(* IEC 61131-3 sources: MyTestRepos/BATTERY/PRG (part 2) *)

(* ---- PRG_DO.st ---- *)
PROGRAM PRG_DO
VAR
	F_Trig : ARRAY[1..cnst_num_do] OF F_TRIG;
	i: INT;
	ManualFixChannels : BOOL; (*Will reset channels if faulty, i.e. card number is zero*)
	Reset: BOOL;
	Firstrun: BOOL;
	(*Interal variables*)
	Fan_SR : 				SR;

	(* Digital Outputs*)
	do_RunningLamp: str_DoProcess;
	do_Running: str_DoProcess;
	do_StoppedLamp: str_DoProcess;
	do_Stopped: str_DoProcess;
	do_FaultLamp: str_DoProcess;
	do_WarningLamp: str_DoProcess;
	do_StartFan: str_DoProcess;
	do_EnergizedLamp: str_DoProcess;
	do_LampTest: str_DoProcess;
	do_ReadyLamp: str_DoProcess;
	do_ChargingLamp: str_DoProcess;
	do_ShutdownPlcFailure: str_DoProcess;
	do_LocalLamp: str_DoProcess;

	do_RunningLamp_daemon: fb_DoProcess;
	do_Running_daemon: fb_DoProcess;
	do_StoppedLamp_daemon: fb_DoProcess;
	do_Stopped_daemon: fb_DoProcess;
	do_FaultLamp_daemon: fb_DoProcess;
	do_WarningLamp_daemon: fb_DoProcess;
	do_StartFan_daemon: fb_DoProcess;
	do_EnergizedLamp_daemon: fb_DoProcess;
	do_LampTest_daemon: fb_DoProcess;
	do_ReadyLamp_daemon: fb_DoProcess;
	do_ChargingLamp_daemon: fb_DoProcess;
	do_ShutdownPlcFailure_daemon: fb_DoProcess;
	do_LocalLamp_daemon: fb_DoProcess;
END_VAR

VAR RETAIN
	do_RunningLamp_setup: str_DoSetup;
	do_Running_setup: str_DoSetup;
	do_StoppedLamp_setup: str_DoSetup;
	do_Stopped_setup: str_DoSetup;
	do_FaultLamp_setup: str_DoSetup;
	do_WarningLamp_setup: str_DoSetup;
	do_StartFan_setup: str_DoSetup;
	do_EnergizedLamp_setup: str_DoSetup;
	do_LampTest_setup: str_DoSetup;
	do_ReadyLamp_setup: str_DoSetup;
	do_ChargingLamp_setup: str_DoSetup;
	do_ShutdownPlcFailure_setup: str_DoSetup;
	do_LocalLamp_setup: str_DoSetup;
END_VAR

Reset := PRG_Functions.Reset;

(*Setup the HMI variables so that they are equal to actual used variables*)
IF (NOT Firstrun) THEN
	hmi_DoSetup[1]:=do_RunningLamp_setup;
	hmi_DoSetup[2]:=do_Running_setup;
	hmi_DoSetup[3]:=do_StoppedLamp_setup;
	hmi_DoSetup[4]:=do_Stopped_setup;
	hmi_DoSetup[5]:=do_FaultLamp_setup;
	hmi_DoSetup[6]:=do_WarningLamp_setup;
	hmi_DoSetup[7]:=do_StartFan_setup;
	hmi_DoSetup[8]:=do_EnergizedLamp_setup;
	hmi_DoSetup[9]:=do_LampTest_setup;
	hmi_DoSetup[10]:=do_ReadyLamp_setup;
	hmi_DoSetup[11]:=do_ChargingLamp_setup;
	hmi_DoSetup[12]:=do_ShutdownPlcFailure_setup;
	hmi_DoSetup[13]:=do_LocalLamp_setup;
	Firstrun := TRUE;
END_IF

do_StartFan_daemon (setup:=do_StartFan_setup,inPV:=do_StartFan);
do_LampTest_daemon (setup:=do_LampTest_setup,inPV:=do_LampTest);
do_Running_daemon (setup:=do_Running_setup,inPV:=do_Running);
do_Stopped_daemon (setup:=do_Stopped_setup,inPV:=do_Stopped);
do_ShutdownPlcFailure_daemon (setup:=do_ShutdownPlcFailure_setup,inPV:=do_ShutdownPlcFailure);

IF PRG_HMI.DoorSettings.enRunningLamp THEN
	do_RunningLamp_daemon (setup:=do_RunningLamp_setup,inPV:=do_RunningLamp);
END_IF

IF PRG_HMI.DoorSettings.enStoppedLamp THEN
	do_StoppedLamp_daemon (setup:=do_StoppedLamp_setup,inPV:=do_StoppedLamp);
END_IF

IF PRG_HMI.DoorSettings.enFaultLamp THEN
	do_FaultLamp_daemon (setup:=do_FaultLamp_setup,inPV:=do_FaultLamp);
END_IF

IF PRG_HMI.DoorSettings.enWarningLamp THEN
	do_WarningLamp_daemon (setup:=do_WarningLamp_setup,inPV:=do_WarningLamp);
END_IF

IF PRG_HMI.DoorSettings.enChargingLamp THEN
	do_ChargingLamp_daemon (setup:=do_ChargingLamp_setup,inPV:=do_ChargingLamp);
END_IF

IF PRG_HMI.DoorSettings.enLocalLamp THEN
	do_LocalLamp_daemon (setup:=do_LocalLamp_setup,inPV:=do_LocalLamp);
END_IF

IF PRG_HMI.DoorSettings.enReadyLamp THEN
	do_ReadyLamp_daemon (setup:=do_ReadyLamp_setup,inPV:=do_ReadyLamp);
END_IF

IF PRG_HMI.DoorSettings.enEnergizedLamp THEN
	do_EnergizedLamp_daemon (setup:=do_EnergizedLamp_setup,inPV:=do_EnergizedLamp);
END_IF

hmi_DoPV[1]:=do_RunningLamp_daemon.inPV;
hmi_DoPV[2]:=do_Running_daemon.inPV;
hmi_DoPV[3]:=do_StoppedLamp_daemon.inPV;
hmi_DoPV[4]:=do_Stopped_daemon.inPV;
hmi_DoPV[5]:=do_FaultLamp_daemon.inPV;
hmi_DoPV[6]:=do_WarningLamp_daemon.inPV;
hmi_DoPV[7]:=do_StartFan_daemon.inPV;
hmi_DoPV[8]:=do_EnergizedLamp_daemon.inPV;
hmi_DoPV[9]:=do_LampTest_daemon.inPV;
hmi_DoPV[10]:=do_ReadyLamp_daemon.inPV;
hmi_DoPV[11]:=do_ChargingLamp_daemon.inPV;
hmi_DoPV[12]:=do_ShutdownPlcFailure_daemon.inPV;
hmi_DoPV[13]:=do_LocalLamp_daemon.inPV;

IF (ManualFixChannels) THEN  (*If manually forced: re-configure the channels*)
	FOR i:=0 TO cnst_num_do BY 1 DO				(*Check if channel info is empty and restore if so.*)
		IF (hmi_DoSetup[i].CardNb = 0 AND PRG_HMI.setup_DioCard1_Number <> 0) THEN
			hmi_RestoreDefault_do[i] := TRUE;
		END_IF
	END_FOR;
	ManualFixChannels := FALSE;
END_IF

(*------------------------------------Control of cabinet lamps -------------------------------------*)

(*In Local Lamp*)
IF PRG_HMI.DoorSettings.enLocalLamp THEN
	IF(PRG_IAS.IasCommunication.Alarm AND (PRG_Operation.ControlPlace.ctrlLocation = e_Remote)) THEN
		do_LocalLamp.PV := PRG_StateMain.LedBlinker.CLK_Pulse;
	ELSE
		do_LocalLamp.PV	:= PRG_Operation.ControlPlace.ctrlLocation = e_Local XOR PRG_HMI.LamptestPulsetrain.CLK_Pulse;
	END_IF
END_IF

(*Running Lamp*)
IF PRG_HMI.DoorSettings.enRunningLamp THEN
	do_RunningLamp.PV := (PRG_StateMain.RunningLamp XOR PRG_HMI.LamptestPulsetrain.CLK_Pulse);
END_IF

(*Stopped Lamp*)
IF PRG_HMI.DoorSettings.enStoppedLamp THEN
	do_StoppedLamp.PV := (PRG_StateMain.StoppedLamp XOR PRG_HMI.LamptestPulsetrain.CLK_Pulse );
END_IF

(*Warning Lamp*)
IF PRG_HMI.DoorSettings.enWarningLamp THEN
	do_WarningLamp.PV := (PRG_Alarms.Repeat_Alarm.Alarm_common XOR PRG_HMI.LamptestPulsetrain.CLK_Pulse);
END_IF

(*Fault Lamp*)
IF PRG_HMI.DoorSettings.enFaultLamp THEN
	do_FaultLamp.PV := (PRG_Faults.Repeat_Fault.Alarm_common XOR PRG_HMI.LamptestPulsetrain.CLK_Pulse);
END_IF

(*Charging Lamp*)
IF PRG_HMI.DoorSettings.enChargingLamp THEN
	do_ChargingLamp.PV := (PRG_Battery.batteryCharging XOR PRG_HMI.LamptestPulsetrain.CLK_Pulse);
END_IF

(*Ready to Start Lamp*)
IF PRG_HMI.DoorSettings.enReadyLamp THEN
	do_ReadyLamp.PV := (PRG_HMI.ReadyToStart XOR PRG_HMI.LamptestPulsetrain.CLK_Pulse);
END_IF

(*Energized Lamp*)
IF PRG_HMI.DoorSettings.enEnergizedLamp THEN
	do_EnergizedLamp.PV := (PRG_Battery.BatteryMinOneConnected XOR PRG_HMI.LamptestPulsetrain.CLK_Pulse);
END_IF

(*Lamp test relay for lamps not connected to PLC*)
do_LampTest.PV := PRG_HMI.LamptestPulsetrain.CLK_Pulse;

(*------------------------------------Hardwire Status Outputs -------------------------------------*)

do_Stopped.PV := PRG_StateMain.StoppedOutput;
do_Running.PV := PRG_StateMain.RunningOutput;

(*------------------------------------Control of cabinet fan -------------------------------------*)
Fan_SR(
	SET1 := PRG_AI.ai_CabinetTemperature.Level.H,
	RESET := PRG_AI.ai_CabinetTemperature.Level.L,
	Q1 => do_StartFan.PV
);

(*------------------------------------ Hardwire Shutdown -------------------------------------*)
(*If modbus fault or no stopping - drop the white gloves.*)
IF 	(PRG_BatteryComm.CorvusBMS_Total_Comm_Fault OR PRG_StateMain.stoppingTON.Q OR PRG_Drive.CommFault[1]) THEN
	do_ShutdownPlcFailure.PV := FALSE;
ELSE
	do_ShutdownPlcFailure.PV := TRUE;
END_IF

END_PROGRAM

ACTIONS

ACTION Settings

(**************do_RunningLamp***********************)
IF (RestoreAllToDefault OR do_RunningLamp_setup.RestoreDefault  OR hmi_RestoreDefault_do[1]) THEN
	do_RunningLamp_setup.Name:='do_RunningLamp';
	do_RunningLamp_setup.CardNb:=PRG_HMI.setup_DioCard1_Number;
	do_RunningLamp_setup.ChannelMode:=2;
	do_RunningLamp_setup.ChannelNb:=1;
	do_RunningLamp_setup.Enable.Forcing:=0;
	do_RunningLamp_setup.Levels.ForceValue:=0;
END_IF
IF (hmi_RestoreDefault_do[1] OR RestoreAllToDefault OR do_RunningLamp_setup.RestoreDefault) THEN (*Copy values into HMI variable and reset*)
	hmi_DoSetup[1]:=do_RunningLamp_setup; (*Copy setup values from retain into hmi variable*)
	hmi_RestoreDefault_do[1]:=FALSE; (*Make sure that the restore variable is turned off after one restore command*)
	do_RunningLamp_setup.RestoreDefault:=FALSE; (*Make sure that the restore variable is turned off after one restore command*)
END_IF
IF (hmi_DoWriteSetup[1]) THEN
	do_RunningLamp_setup:=hmi_DoSetup[1]; (*Paste hmi changes back into setup variable*)
	hmi_DoWriteSetup[1]:=FALSE; (*Make sure that the write variable is turned off after one write command*)
END_IF
F_Trig[1](CLK:=hmi_DoPV[1].IsForced); (*Reset HMI forcing dialog when timer runs out*)
IF (F_Trig[1].Q) THEN hmi_DoSetup[1].Enable.Forcing:=FALSE;do_RunningLamp_setup.Enable.Forcing:=FALSE; END_IF
(**************************************************)

(**************do_Running***********************)
IF (RestoreAllToDefault OR do_Running_setup.RestoreDefault  OR hmi_RestoreDefault_do[2]) THEN
	do_Running_setup.Name:='do_Running';
	do_Running_setup.CardNb:=PRG_HMI.setup_DioCard1_Number;
	do_Running_setup.ChannelMode:=2;
	do_Running_setup.ChannelNb:=2;
	do_Running_setup.Enable.Forcing:=0;
	do_Running_setup.Levels.ForceValue:=0;
END_IF
IF (hmi_RestoreDefault_do[2] OR RestoreAllToDefault OR do_Running_setup.RestoreDefault) THEN (*Copy values into HMI variable and reset*)
	hmi_DoSetup[2]:=do_Running_setup; (*Copy setup values from retain into hmi variable*)
	hmi_RestoreDefault_do[2]:=FALSE; (*Make sure that the restore variable is turned off after one restore command*)
	do_Running_setup.RestoreDefault:=FALSE; (*Make sure that the restore variable is turned off after one restore command*)
END_IF
IF (hmi_DoWriteSetup[2]) THEN
	do_Running_setup:=hmi_DoSetup[2]; (*Paste hmi changes back into setup variable*)
	hmi_DoWriteSetup[2]:=FALSE; (*Make sure that the write variable is turned off after one write command*)
END_IF
F_Trig[2](CLK:=hmi_DoPV[2].IsForced); (*Reset HMI forcing dialog when timer runs out*)
IF (F_Trig[2].Q) THEN hmi_DoSetup[2].Enable.Forcing:=FALSE;do_Running_setup.Enable.Forcing:=FALSE; END_IF
(**************************************************)

(**************do_StoppedLamp***********************)
IF (RestoreAllToDefault OR do_StoppedLamp_setup.RestoreDefault  OR hmi_RestoreDefault_do[3]) THEN
	do_StoppedLamp_setup.Name:='do_StoppedLamp';
	do_StoppedLamp_setup.CardNb:=PRG_HMI.setup_DioCard1_Number;
	do_StoppedLamp_setup.ChannelMode:=2;
	do_StoppedLamp_setup.ChannelNb:=3;
	do_StoppedLamp_setup.Enable.Forcing:=0;
	do_StoppedLamp_setup.Levels.ForceValue:=0;
END_IF
IF (hmi_RestoreDefault_do[3] OR RestoreAllToDefault OR do_StoppedLamp_setup.RestoreDefault) THEN (*Copy values into HMI variable and reset*)
	hmi_DoSetup[3]:=do_StoppedLamp_setup; (*Copy setup values from retain into hmi variable*)
	hmi_RestoreDefault_do[3]:=FALSE; (*Make sure that the restore variable is turned off after one restore command*)
	do_StoppedLamp_setup.RestoreDefault:=FALSE; (*Make sure that the restore variable is turned off after one restore command*)
END_IF
IF (hmi_DoWriteSetup[3]) THEN
	do_StoppedLamp_setup:=hmi_DoSetup[3]; (*Paste hmi changes back into setup variable*)
	hmi_DoWriteSetup[3]:=FALSE; (*Make sure that the write variable is turned off after one write command*)
END_IF
F_Trig[3](CLK:=hmi_DoPV[3].IsForced); (*Reset HMI forcing dialog when timer runs out*)
IF (F_Trig[3].Q) THEN hmi_DoSetup[3].Enable.Forcing:=FALSE;do_StoppedLamp_setup.Enable.Forcing:=FALSE; END_IF
(**************************************************)

(**************do_Stopped***********************)
IF (RestoreAllToDefault OR do_Stopped_setup.RestoreDefault  OR hmi_RestoreDefault_do[4]) THEN
	do_Stopped_setup.Name:='do_Stopped';
	do_Stopped_setup.CardNb:=PRG_HMI.setup_DioCard1_Number;
	do_Stopped_setup.ChannelMode:=2;
	do_Stopped_setup.ChannelNb:=4;
	do_Stopped_setup.Enable.Forcing:=0;
	do_Stopped_setup.Levels.ForceValue:=0;
END_IF
IF (hmi_RestoreDefault_do[4] OR RestoreAllToDefault OR do_Stopped_setup.RestoreDefault) THEN (*Copy values into HMI variable and reset*)
	hmi_DoSetup[4]:=do_Stopped_setup; (*Copy setup values from retain into hmi variable*)
	hmi_RestoreDefault_do[4]:=FALSE; (*Make sure that the restore variable is turned off after one restore command*)
	do_Stopped_setup.RestoreDefault:=FALSE; (*Make sure that the restore variable is turned off after one restore command*)
END_IF
IF (hmi_DoWriteSetup[4]) THEN
	do_Stopped_setup:=hmi_DoSetup[4]; (*Paste hmi changes back into setup variable*)
	hmi_DoWriteSetup[4]:=FALSE; (*Make sure that the write variable is turned off after one write command*)
END_IF
F_Trig[4](CLK:=hmi_DoPV[4].IsForced); (*Reset HMI forcing dialog when timer runs out*)
IF (F_Trig[4].Q) THEN hmi_DoSetup[4].Enable.Forcing:=FALSE;do_Stopped_setup.Enable.Forcing:=FALSE; END_IF
(**************************************************)

(**************do_FaultLamp***********************)
IF (RestoreAllToDefault OR do_FaultLamp_setup.RestoreDefault  OR hmi_RestoreDefault_do[5]) THEN
	do_FaultLamp_setup.Name:='do_FaultLamp';
	do_FaultLamp_setup.CardNb:=PRG_HMI.setup_DioCard1_Number;
	do_FaultLamp_setup.ChannelMode:=2;
	do_FaultLamp_setup.ChannelNb:=5;
	do_FaultLamp_setup.Enable.Forcing:=0;
	do_FaultLamp_setup.Levels.ForceValue:=0;
END_IF
IF (hmi_RestoreDefault_do[5] OR RestoreAllToDefault OR do_FaultLamp_setup.RestoreDefault) THEN (*Copy values into HMI variable and reset*)
	hmi_DoSetup[5]:=do_FaultLamp_setup; (*Copy setup values from retain into hmi variable*)
	hmi_RestoreDefault_do[5]:=FALSE; (*Make sure that the restore variable is turned off after one restore command*)
	do_FaultLamp_setup.RestoreDefault:=FALSE; (*Make sure that the restore variable is turned off after one restore command*)
END_IF
IF (hmi_DoWriteSetup[5]) THEN
	do_FaultLamp_setup:=hmi_DoSetup[5]; (*Paste hmi changes back into setup variable*)
	hmi_DoWriteSetup[5]:=FALSE; (*Make sure that the write variable is turned off after one write command*)
END_IF
F_Trig[5](CLK:=hmi_DoPV[5].IsForced); (*Reset HMI forcing dialog when timer runs out*)
IF (F_Trig[5].Q) THEN hmi_DoSetup[5].Enable.Forcing:=FALSE;do_FaultLamp_setup.Enable.Forcing:=FALSE; END_IF
(**************************************************)

(**************do_WarningLamp***********************)
IF (RestoreAllToDefault OR do_WarningLamp_setup.RestoreDefault  OR hmi_RestoreDefault_do[6]) THEN
	do_WarningLamp_setup.Name:='do_WarningLamp';
	do_WarningLamp_setup.CardNb:=PRG_HMI.setup_DioCard1_Number;
	do_WarningLamp_setup.ChannelMode:=2;
	do_WarningLamp_setup.ChannelNb:=6;
	do_WarningLamp_setup.Enable.Forcing:=0;
	do_WarningLamp_setup.Levels.ForceValue:=0;
END_IF
IF (hmi_RestoreDefault_do[6] OR RestoreAllToDefault OR do_WarningLamp_setup.RestoreDefault) THEN (*Copy values into HMI variable and reset*)
	hmi_DoSetup[6]:=do_WarningLamp_setup; (*Copy setup values from retain into hmi variable*)
	hmi_RestoreDefault_do[6]:=FALSE; (*Make sure that the restore variable is turned off after one restore command*)
	do_WarningLamp_setup.RestoreDefault:=FALSE; (*Make sure that the restore variable is turned off after one restore command*)
END_IF
IF (hmi_DoWriteSetup[6]) THEN
	do_WarningLamp_setup:=hmi_DoSetup[6]; (*Paste hmi changes back into setup variable*)
	hmi_DoWriteSetup[6]:=FALSE; (*Make sure that the write variable is turned off after one write command*)
END_IF
F_Trig[6](CLK:=hmi_DoPV[6].IsForced); (*Reset HMI forcing dialog when timer runs out*)
IF (F_Trig[6].Q) THEN hmi_DoSetup[6].Enable.Forcing:=FALSE;do_WarningLamp_setup.Enable.Forcing:=FALSE; END_IF
(**************************************************)

(**************do_StartFan***********************)
IF (RestoreAllToDefault OR do_StartFan_setup.RestoreDefault  OR hmi_RestoreDefault_do[7]) THEN
	do_StartFan_setup.Name:='do_StartFan';
	do_StartFan_setup.CardNb:=PRG_HMI.setup_DioCard1_Number;
	do_StartFan_setup.ChannelMode:=2;
	do_StartFan_setup.ChannelNb:=10;
	do_StartFan_setup.Enable.Forcing:=0;
	do_StartFan_setup.Levels.ForceValue:=0;
END_IF
IF (hmi_RestoreDefault_do[7] OR RestoreAllToDefault OR do_StartFan_setup.RestoreDefault) THEN (*Copy values into HMI variable and reset*)
	hmi_DoSetup[7]:=do_StartFan_setup; (*Copy setup values from retain into hmi variable*)
	hmi_RestoreDefault_do[7]:=FALSE; (*Make sure that the restore variable is turned off after one restore command*)
	do_StartFan_setup.RestoreDefault:=FALSE; (*Make sure that the restore variable is turned off after one restore command*)
END_IF
IF (hmi_DoWriteSetup[7]) THEN
	do_StartFan_setup:=hmi_DoSetup[7]; (*Paste hmi changes back into setup variable*)
	hmi_DoWriteSetup[7]:=FALSE; (*Make sure that the write variable is turned off after one write command*)
END_IF
F_Trig[7](CLK:=hmi_DoPV[7].IsForced); (*Reset HMI forcing dialog when timer runs out*)
IF (F_Trig[7].Q) THEN hmi_DoSetup[7].Enable.Forcing:=FALSE;do_StartFan_setup.Enable.Forcing:=FALSE; END_IF
(**************************************************)

(**************do_EnergizedLamp***********************)
IF (RestoreAllToDefault OR do_EnergizedLamp_setup.RestoreDefault  OR hmi_RestoreDefault_do[8]) THEN
	do_EnergizedLamp_setup.Name:='do_EnergizedLamp';
	do_EnergizedLamp_setup.CardNb:=PRG_HMI.setup_DioCard1_Number;
	do_EnergizedLamp_setup.ChannelMode:=2;
	do_EnergizedLamp_setup.ChannelNb:=11;
	do_EnergizedLamp_setup.Enable.Forcing:=0;
	do_EnergizedLamp_setup.Levels.ForceValue:=0;
END_IF
IF (hmi_RestoreDefault_do[8] OR RestoreAllToDefault OR do_EnergizedLamp_setup.RestoreDefault) THEN (*Copy values into HMI variable and reset*)
	hmi_DoSetup[8]:=do_EnergizedLamp_setup; (*Copy setup values from retain into hmi variable*)
	hmi_RestoreDefault_do[8]:=FALSE; (*Make sure that the restore variable is turned off after one restore command*)
	do_EnergizedLamp_setup.RestoreDefault:=FALSE; (*Make sure that the restore variable is turned off after one restore command*)
END_IF
IF (hmi_DoWriteSetup[8]) THEN
	do_EnergizedLamp_setup:=hmi_DoSetup[8]; (*Paste hmi changes back into setup variable*)
	hmi_DoWriteSetup[8]:=FALSE; (*Make sure that the write variable is turned off after one write command*)
END_IF
F_Trig[8](CLK:=hmi_DoPV[8].IsForced); (*Reset HMI forcing dialog when timer runs out*)
IF (F_Trig[8].Q) THEN hmi_DoSetup[8].Enable.Forcing:=FALSE;do_EnergizedLamp_setup.Enable.Forcing:=FALSE; END_IF
(**************************************************)

(**************do_LampTest***********************)
IF (RestoreAllToDefault OR do_LampTest_setup.RestoreDefault  OR hmi_RestoreDefault_do[9]) THEN
	do_LampTest_setup.Name:='do_LampTest';
	do_LampTest_setup.CardNb:=PRG_HMI.setup_DioCard1_Number;
	do_LampTest_setup.ChannelMode:=2;
	do_LampTest_setup.ChannelNb:=12;
	do_LampTest_setup.Enable.Forcing:=0;
	do_LampTest_setup.Levels.ForceValue:=0;
END_IF
IF (hmi_RestoreDefault_do[9] OR RestoreAllToDefault OR do_LampTest_setup.RestoreDefault) THEN (*Copy values into HMI variable and reset*)
	hmi_DoSetup[9]:=do_LampTest_setup; (*Copy setup values from retain into hmi variable*)
	hmi_RestoreDefault_do[9]:=FALSE; (*Make sure that the restore variable is turned off after one restore command*)
	do_LampTest_setup.RestoreDefault:=FALSE; (*Make sure that the restore variable is turned off after one restore command*)
END_IF
IF (hmi_DoWriteSetup[9]) THEN
	do_LampTest_setup:=hmi_DoSetup[9]; (*Paste hmi changes back into setup variable*)
	hmi_DoWriteSetup[9]:=FALSE; (*Make sure that the write variable is turned off after one write command*)
END_IF
F_Trig[9](CLK:=hmi_DoPV[9].IsForced); (*Reset HMI forcing dialog when timer runs out*)
IF (F_Trig[9].Q) THEN hmi_DoSetup[9].Enable.Forcing:=FALSE;do_LampTest_setup.Enable.Forcing:=FALSE; END_IF
(**************************************************)

(**************do_ReadyLamp***********************)
IF (RestoreAllToDefault OR do_ReadyLamp_setup.RestoreDefault  OR hmi_RestoreDefault_do[10]) THEN
	do_ReadyLamp_setup.Name:='do_ReadyLamp';
	do_ReadyLamp_setup.CardNb:=PRG_HMI.setup_DioCard1_Number;
	do_ReadyLamp_setup.ChannelMode:=2;
	do_ReadyLamp_setup.ChannelNb:=13;
	do_ReadyLamp_setup.Enable.Forcing:=0;
	do_ReadyLamp_setup.Levels.ForceValue:=0;
END_IF
IF (hmi_RestoreDefault_do[10] OR RestoreAllToDefault OR do_ReadyLamp_setup.RestoreDefault) THEN (*Copy values into HMI variable and reset*)
	hmi_DoSetup[10]:=do_ReadyLamp_setup; (*Copy setup values from retain into hmi variable*)
	hmi_RestoreDefault_do[10]:=FALSE; (*Make sure that the restore variable is turned off after one restore command*)
	do_ReadyLamp_setup.RestoreDefault:=FALSE; (*Make sure that the restore variable is turned off after one restore command*)
END_IF
IF (hmi_DoWriteSetup[10]) THEN
	do_ReadyLamp_setup:=hmi_DoSetup[10]; (*Paste hmi changes back into setup variable*)
	hmi_DoWriteSetup[10]:=FALSE; (*Make sure that the write variable is turned off after one write command*)
END_IF
F_Trig[10](CLK:=hmi_DoPV[10].IsForced); (*Reset HMI forcing dialog when timer runs out*)
IF (F_Trig[10].Q) THEN hmi_DoSetup[10].Enable.Forcing:=FALSE;do_ReadyLamp_setup.Enable.Forcing:=FALSE; END_IF
(**************************************************)

(**************do_ChargingLamp***********************)
IF (RestoreAllToDefault OR do_ChargingLamp_setup.RestoreDefault  OR hmi_RestoreDefault_do[11]) THEN
	do_ChargingLamp_setup.Name:='do_ChargingLamp';
	do_ChargingLamp_setup.CardNb:=PRG_HMI.setup_DioCard1_Number;
	do_ChargingLamp_setup.ChannelMode:=2;
	do_ChargingLamp_setup.ChannelNb:=14;
	do_ChargingLamp_setup.Enable.Forcing:=0;
	do_ChargingLamp_setup.Levels.ForceValue:=0;
END_IF
IF (hmi_RestoreDefault_do[11] OR RestoreAllToDefault OR do_ChargingLamp_setup.RestoreDefault) THEN (*Copy values into HMI variable and reset*)
	hmi_DoSetup[11]:=do_ChargingLamp_setup; (*Copy setup values from retain into hmi variable*)
	hmi_RestoreDefault_do[11]:=FALSE; (*Make sure that the restore variable is turned off after one restore command*)
	do_ChargingLamp_setup.RestoreDefault:=FALSE; (*Make sure that the restore variable is turned off after one restore command*)
END_IF
IF (hmi_DoWriteSetup[11]) THEN
	do_ChargingLamp_setup:=hmi_DoSetup[11]; (*Paste hmi changes back into setup variable*)
	hmi_DoWriteSetup[11]:=FALSE; (*Make sure that the write variable is turned off after one write command*)
END_IF
F_Trig[11](CLK:=hmi_DoPV[11].IsForced); (*Reset HMI forcing dialog when timer runs out*)
IF (F_Trig[11].Q) THEN hmi_DoSetup[11].Enable.Forcing:=FALSE;do_ChargingLamp_setup.Enable.Forcing:=FALSE; END_IF
(**************************************************)

(**************do_ShutdownPlcFailure***********************)
IF (RestoreAllToDefault OR do_ShutdownPlcFailure_setup.RestoreDefault  OR hmi_RestoreDefault_do[12]) THEN
	do_ShutdownPlcFailure_setup.Name:='do_ShutdownPlcFailure';
	do_ShutdownPlcFailure_setup.CardNb:=PRG_HMI.setup_DioCard1_Number;
	do_ShutdownPlcFailure_setup.ChannelMode:=2;
	do_ShutdownPlcFailure_setup.ChannelNb:=15;
	do_ShutdownPlcFailure_setup.Enable.Forcing:=0;
	do_ShutdownPlcFailure_setup.Levels.ForceValue:=0;
END_IF
IF (hmi_RestoreDefault_do[12] OR RestoreAllToDefault OR do_ShutdownPlcFailure_setup.RestoreDefault) THEN (*Copy values into HMI variable and reset*)
	hmi_DoSetup[12]:=do_ShutdownPlcFailure_setup; (*Copy setup values from retain into hmi variable*)
	hmi_RestoreDefault_do[12]:=FALSE; (*Make sure that the restore variable is turned off after one restore command*)
	do_ShutdownPlcFailure_setup.RestoreDefault:=FALSE; (*Make sure that the restore variable is turned off after one restore command*)
END_IF
IF (hmi_DoWriteSetup[12]) THEN
	do_ShutdownPlcFailure_setup:=hmi_DoSetup[12]; (*Paste hmi changes back into setup variable*)
	hmi_DoWriteSetup[12]:=FALSE; (*Make sure that the write variable is turned off after one write command*)
END_IF
F_Trig[12](CLK:=hmi_DoPV[12].IsForced); (*Reset HMI forcing dialog when timer runs out*)
IF (F_Trig[12].Q) THEN hmi_DoSetup[12].Enable.Forcing:=FALSE;do_ShutdownPlcFailure_setup.Enable.Forcing:=FALSE; END_IF
(**************************************************)

(**************do_LocalLamp***********************)
IF (RestoreAllToDefault OR do_LocalLamp_setup.RestoreDefault  OR hmi_RestoreDefault_do[13]) THEN
	do_LocalLamp_setup.Name:='do_LocalLamp';
	do_LocalLamp_setup.CardNb:=PRG_HMI.setup_DioCard1_Number;
	do_LocalLamp_setup.ChannelMode:=2;
	do_LocalLamp_setup.ChannelNb:=16;
	do_LocalLamp_setup.Enable.Forcing:=0;
	do_LocalLamp_setup.Levels.ForceValue:=0;
END_IF
IF (hmi_RestoreDefault_do[13] OR RestoreAllToDefault OR do_LocalLamp_setup.RestoreDefault) THEN (*Copy values into HMI variable and reset*)
	hmi_DoSetup[13]:=do_LocalLamp_setup; (*Copy setup values from retain into hmi variable*)
	hmi_RestoreDefault_do[13]:=FALSE; (*Make sure that the restore variable is turned off after one restore command*)
	do_LocalLamp_setup.RestoreDefault:=FALSE; (*Make sure that the restore variable is turned off after one restore command*)
END_IF
IF (hmi_DoWriteSetup[13]) THEN
	do_LocalLamp_setup:=hmi_DoSetup[13]; (*Paste hmi changes back into setup variable*)
	hmi_DoWriteSetup[13]:=FALSE; (*Make sure that the write variable is turned off after one write command*)
END_IF
F_Trig[13](CLK:=hmi_DoPV[13].IsForced); (*Reset HMI forcing dialog when timer runs out*)
IF (F_Trig[13].Q) THEN hmi_DoSetup[13].Enable.Forcing:=FALSE;do_LocalLamp_setup.Enable.Forcing:=FALSE; END_IF
(**************************************************)

END_ACTION

END_ACTIONS

(* ---- PRG_Drive.st ---- *)
PROGRAM PRG_Drive
VAR
	(*Unit over temp alarm*)
	UnitOverTempTON : 		TON; (*Timer with time delay for over temperature alarm*)
	UnitOverTempAlarm : 	BOOL; (*Vacon unit is over heated*)

	(*Vacon Data variables*)
	Profinet_IO	:	ARRAY[1..4] OF pnVaconIO;		(*Function block handling IO to and from Vacon Profidrive*)
	CW :			str_VaconCW_DcDc;					(*Command word to vacon*)
	CommandWord :	DINT;								(*Command word in DINT format to Vacon*)
	SW :			ARRAY[1..4] OF str_VaconSW_DcDc;	(*Standard FB status word ID68 + extended application status word ID43*)
	StatusWord:		ARRAY[1..4] OF fb_BitToWord;		(*Status Word*)
	FW :			ARRAY[1..4] OF str_VaconFW_DcDc;	(*Fault Word 1*)
	FW2 :			ARRAY[1..4] OF str_VaconFW2_DcDc;	(*Fault Word 2*)
	PDO :			ARRAY[1..4] OF str_VaconPDO_DcDc;	(*Analog data from vacon in engineering and perunit values*)
	PDI :			ARRAY[1..4] OF str_VaconPDI_DcDc; 	(*Analog values prepared for transmittal to Vacon*)

	(*Watchdog and comm faults*)
	Watchdog:				ARRAY[1..4] OF pnVaconWD;
	Watchdog_Setup:			str_VaconWd;
	CommFault :				ARRAY[1..4] OF BOOL;

	i : INT; (*Looping variable*)

	(*Analog Values from Vacon Drives*)
	Data:				str_DriveData_DcDc; 	(*Formatted values in per-unit or engineering values from drive*)
	Status:				str_DriveStatus_DcDc; 	(*Status word from master drive*)

	(*Misc*)
	StartStop: 				RS;
	StartTON: 				TON;
END_VAR

(*
 * =======================================================================================================================================
 * Raw information to and from Vacon ProfiDrive
 * =======================================================================================================================================
*)
Profinet_IO[1](
 	(*Commands and references to Vacon*)
	CW := CommandWord,						(*ID1160 FB Control Word*)
	Ref := PDI[1].Ref,						(*Reference not in use*)
	PDI_1 := PDI[1].PDI1_UndervoltageRef ,	(*ID1567: Under Voltage Reference *)
	PDI_2 := PDI[1].PDI2_OvervoltageRef ,	(*ID1528: Over Voltage Reference*)
	PDI_3 := PDI[1].PDI3_ChargeLimit ,		(*ID1290: Charging current limit in percentage of Source Nom Current *)
	PDI_4 := PDI[1].PDI4_DischargeLimit ,	(*ID1289: Discharging current limit in percentage of Source Nom Current *)
	PDI_5 := PDI[1].PDI5_SourceMaxVoltage ,	(*ID1895: Source Max Voltage*)
	PDI_6 := PDI[1].PDI6_SourceMinVoltage ,	(*ID1893: Source Min Voltage*)
	PDI_7 := 0,
	PDI_8 := 0,
	moduleNr := PRG_HMI.setup_Drive_PnMasterCardNr[1],

	(*Status and values from Vacon*)
	SW =>  ,									(*ID68: Fieldbus Status Word*)
	ACT => PDO[1].ACT_DcLinkVoltage_eng ,		(*Feedback DC Link Voltage*)
	PDO_1 => PDO[1].PDO1_ActiveCurrent_pu ,		(*ID1125: Active Current*)
	PDO_2 => PDO[1].PDO2_SourcePower_pu ,		(*ID5: Source Power *)
	PDO_3 => PDO[1].PDO3_SourceVoltage_eng ,	(*ID1107: Source Voltage*)
	PDO_4 => PDO[1].PDO4_SW43 ,					(*ID43: Application Specific Status Word*)
	PDO_5 => PDO[1].PDO5_UnitTemp_eng ,			(*ID1109: Unit Temperature*)
	PDO_6 => PDO[1].PDO6_UsedDischargeLimit_pu,	(*ID1855: Discharge Limit*)
	PDO_7 => PDO[1].PDO7_FaultWord2DcDc,		(*ID1173: Fault Word 2*)
	PDO_8 => PDO[1].PDO8_FaultWordDcDc ,		(*ID1172: Fault Word 1*)
	mioGetError => ,
	mioSetError =>
);

(*
 * =======================================================================================================================================
 * Set Status Words
 * =======================================================================================================================================
*)

(*General Part from ID68*)
SW[1].b0_ReadyOn := 			Profinet_IO[1].SW.0;	(*Drive ready to start charging *)
SW[1].b1_ReadyRun := 			Profinet_IO[1].SW.1;	(*Drive ready and Main Contactor is ON*)
SW[1].b2_Running := 			Profinet_IO[1].SW.2;	(*Drive in Run state (Modulating)*)
SW[1].b3_Fault := 				Profinet_IO[1].SW.3;	(*Fault is active*)
SW[1].b4_RunEnable := 			Profinet_IO[1].SW.4;	(*Run Enabled. Drive can be started.*)
SW[1].b5_Spare := 				Profinet_IO[1].SW.5; 	(*Bit 5 NOT in use*)
SW[1].b6_Inhibit := 			Profinet_IO[1].SW.6;	(*Run disabled or fault state.*)
SW[1].b7_Warning := 			Profinet_IO[1].SW.7;	(*Warning active*)
SW[1].b8_Spare := 				Profinet_IO[1].SW.8;	(*Bit 8 NOT in use*)
SW[1].b9_FieldbusCtrlActive := 	Profinet_IO[1].SW.9;	(*Fieldbus control active  *)
SW[1].b10_Spare := 				Profinet_IO[1].SW.10;	(*Bit 10 NOT in use*)
SW[1].b11_Spare := 				Profinet_IO[1].SW.11;	(*Bit 11 NOT in use*)
SW[1].b12_Spare := 				Profinet_IO[1].SW.12;	(*Bit 12 NOT in use*)
SW[1].b13_Spare := 				Profinet_IO[1].SW.13;	(*Bit 13 NOT in use*)
SW[1].b14_Spare := 				Profinet_IO[1].SW.14;	(*Bit 14 NOT in use*)
SW[1].b15_WatchdogPulse := 		Profinet_IO[1].SW.15;	(*Same as received on bit 11 of the main control word.*)

(*Application Specific Status Word ID43*)
SW[1].app.b0_ClosedLoopActive := 	PDO[1].PDO4_SW43.0;		(*Closed Loop Control active *)
SW[1].app.b1_Ready := 				PDO[1].PDO4_SW43.1;		(*Drive in ready state, start command can be given. *)
SW[1].app.b2_Running:= 				PDO[1].PDO4_SW43.2;		(*Drive is modulating. *)
SW[1].app.b3_Fault := 				PDO[1].PDO4_SW43.3;		(*Drive has active faults.*)
SW[1].app.b4_DischargeAllowed := 	PDO[1].PDO4_SW43.4;		(*Discharging allowed*)
SW[1].app.b5_ChargeAllowed := 		PDO[1].PDO4_SW43.5;		(*Charging allowed*)
SW[1].app.b6_RunEnable := 			PDO[1].PDO4_SW43.6;		(*Run Enable command to motor control is high. *)
SW[1].app.b7_Warning := 			PDO[1].PDO4_SW43.7;		(*Drive has active warning signal. Warning signal not stop the operation.*)
SW[1].app.b8_ChargeSwitchClosed :=	PDO[1].PDO4_SW43.8;		(*DC voltage level is above closing limit and no interlock active internally. *)
SW[1].app.b9_OverVoltRegActive := 	PDO[1].PDO4_SW43.9;		(*Over Voltage Regulator Active*)
SW[1].app.b10_UnderVoltRegActive :=	PDO[1].PDO4_SW43.10;	(*Under Voltage Regulator Active*)
SW[1].app.b11_Spare := 				PDO[1].PDO4_SW43.11;	(*Not In Use*)
SW[1].app.b12_RunRequest := 		PDO[1].PDO4_SW43.12;	(*Run Request*)
SW[1].app.b13_RegulatorsActive := 	PDO[1].PDO4_SW43.13;	(*One or more regulators active*)
SW[1].app.b14_VoltageCtrlMode := 	PDO[1].PDO4_SW43.14;	(*Voltage Control Mode*)
SW[1].app.b15_Spare := 				PDO[1].PDO4_SW43.15;	(*Not In Use*)

(*
 * =======================================================================================================================================
 * Watchdog
 * =======================================================================================================================================
*)

Watchdog[1](
	Puls_IN	  := SW[1].b15_WatchdogPulse,
	inVacon	  := Watchdog_Setup,
	Reset  	  := PRG_Functions.Reset,
	Puls_OUT  => ,
	Alarm	  =>,
	AlarmAuto =>
);

CommFault[1] := ((Profinet_IO[1].mioGetError <> 0) OR (Profinet_IO[1].mioSetError <> 0) OR Watchdog[1].AlarmAuto);

(*
 * =======================================================================================================================================
 * Explode Fault Word
 * =======================================================================================================================================
*)

(*Feedback Fault Word*)
FW[1].b0_F1_Overcurrent := 			PDO[1].PDO8_FaultWordDcDc.0;
FW[1].b1_F2_OverVoltage  := 		PDO[1].PDO8_FaultWordDcDc.1;
FW[1].b2_F9_UnderVoltage := 		PDO[1].PDO8_FaultWordDcDc.2;
FW[1].b3_Spare :=					PDO[1].PDO8_FaultWordDcDc.3;
FW[1].b4_F3_EarthFaultDrive :=		PDO[1].PDO8_FaultWordDcDc.4;
FW[1].b5_Spare :=					PDO[1].PDO8_FaultWordDcDc.5;
FW[1].b6_F14_UnitOverTemp :=		PDO[1].PDO8_FaultWordDcDc.6;
FW[1].b7_F29_ThermistorFault :=		PDO[1].PDO8_FaultWordDcDc.7;
FW[1].b8_Spare :=					PDO[1].PDO8_FaultWordDcDc.8;
FW[1].b9_Spare :=					PDO[1].PDO8_FaultWordDcDc.9;
FW[1].b10_Spare :=					PDO[1].PDO8_FaultWordDcDc.10;
FW[1].b11_F52_KeypadCommFault := 	PDO[1].PDO8_FaultWordDcDc.11;
FW[1].b12_F53_FieldbusCommFault := 	PDO[1].PDO8_FaultWordDcDc.12;
FW[1].b13_Spare := 					PDO[1].PDO8_FaultWordDcDc.13;
FW[1].b14_F54_SlotCommFault := 		PDO[1].PDO8_FaultWordDcDc.14;
FW[1].b15_F50_4mAFault := 			PDO[1].PDO8_FaultWordDcDc.15;

FW2[1].b0_F11_OutputPhase :=	PDO[1].PDO7_FaultWord2DcDc.0;
FW2[1].b6_F51_ExternalFault :=	PDO[1].PDO7_FaultWord2DcDc.6;
FW2[1].b9_F31_F41_IGBT :=		PDO[1].PDO7_FaultWord2DcDc.9;
FW2[1].b14_F64_MainSwitchStateFault :=	PDO[1].PDO7_FaultWord2DcDc.14;

(*
 * =======================================================================================================================================
 * Write Command Word
 * =======================================================================================================================================
*)
CommandWord.0 := 	CW.b0_DcChargeContactor := 	StartStop.Q1;
CommandWord.3 := 	CW.b3_Start := 				StartTON.Q;
CommandWord.7 := 	CW.b7_Reset :=				PRG_Functions.Reset;
CommandWord.10 := 	CW.b10_FieldbusCtrl :=		TRUE;
CommandWord.11 := 	CW.b11_Watchdog :=			Watchdog[1].Puls_OUT;

(*
 * =======================================================================================================================================
 * Translate analog data FROM vacon to per unit or engineering values
 * =======================================================================================================================================
*)

(*DC Link Voltage in Volt*)
Data.DcLinkVoltage_eng := PDO[1].ACT_DcLinkVoltage_eng;

(*Current to Source in Amp*)
Data.SourceCurrent_eng[1] := fun_U2S(PDO[1].PDO1_ActiveCurrent_pu) * PRG_HMI.DriveSettings.SourceNomCurrent/1000;
Data.SourceCurrent_eng[2] := fun_U2S(PDO[2].PDO1_ActiveCurrent_pu) * PRG_HMI.DriveSettings.SourceNomCurrent/1000;
Data.SourceCurrent_eng[3] := fun_U2S(PDO[3].PDO1_ActiveCurrent_pu) * PRG_HMI.DriveSettings.SourceNomCurrent/1000;
Data.SourceCurrent_eng[4] := fun_U2S(PDO[4].PDO1_ActiveCurrent_pu) * PRG_HMI.DriveSettings.SourceNomCurrent/1000;

Data.SourceCurrentTotal_eng := (Data.SourceCurrent_eng[1]
 							+	Data.SourceCurrent_eng[2]
 							+	Data.SourceCurrent_eng[3]
 							+	Data.SourceCurrent_eng[4]
							);

(*Power to Source in per-unit of source nominal power and kW*)
Data.SourcePower_pu[1] := fun_U2S(PDO[1].PDO2_SourcePower_pu)/1000 ;
Data.SourcePower_pu[2] := fun_U2S(PDO[2].PDO2_SourcePower_pu)/1000 ;
Data.SourcePower_pu[3] := fun_U2S(PDO[3].PDO2_SourcePower_pu)/1000 ;
Data.SourcePower_pu[4] := fun_U2S(PDO[4].PDO2_SourcePower_pu)/1000 ;

Data.SourcePower_eng[1] := Data.SourcePower_pu[1] * PRG_HMI.DriveSettings.SourceNomPower;
Data.SourcePower_eng[2] := Data.SourcePower_pu[2] * PRG_HMI.DriveSettings.SourceNomPower;
Data.SourcePower_eng[3] := Data.SourcePower_pu[3] * PRG_HMI.DriveSettings.SourceNomPower;
Data.SourcePower_eng[4] := Data.SourcePower_pu[4] * PRG_HMI.DriveSettings.SourceNomPower;

Data.SourcePowerTotal_eng := (	Data.SourcePower_eng[1]
 							+ 	Data.SourcePower_eng[2]
 							+ 	Data.SourcePower_eng[3]
 							+ 	Data.SourcePower_eng[4]
 								);

(*Source Voltage in Volt*)
Data.SourceVoltage_eng := DINT_TO_REAL(PDO[1].PDO3_SourceVoltage_eng)/10;

(*Unit Temperature in °C*)
Data.UnitTemp_eng[1] :=  DINT_TO_REAL(PDO[1].PDO5_UnitTemp_eng);
Data.UnitTemp_eng[2] :=  DINT_TO_REAL(PDO[2].PDO5_UnitTemp_eng);
Data.UnitTemp_eng[3] :=  DINT_TO_REAL(PDO[3].PDO5_UnitTemp_eng);
Data.UnitTemp_eng[4] :=  DINT_TO_REAL(PDO[4].PDO5_UnitTemp_eng);

Data.UnitTempMax_eng := MAX(MAX(MAX(Data.UnitTemp_eng[1], Data.UnitTemp_eng[2]),Data.UnitTemp_eng[3]),Data.UnitTemp_eng[4]);

(*Used Charge and Discharge Limit in per-unit of source nominal current and Ampere*)
Data.UsedDischargeLimit_pu := 	DINT_TO_REAL(PDO[1].PDO6_UsedDischargeLimit_pu)/100;
Data.UsedDischargeLimit_eng := 	fun_SafeDivide(divident := Data.UsedDischargeLimit_pu, devisor := PRG_HMI.DriveSettings.SourceNomCurrent);
Data.UsedChargeLimit_eng := 	fun_SafeDivide(divident := Data.UsedChargeLimit_pu, devisor := PRG_HMI.DriveSettings.SourceNomCurrent);

(*
 * =======================================================================================================================================
 * Set status word from Master drive
 * =======================================================================================================================================
*)

(*General Feedback statuses*)
Status.ReadyOn := 	SW[1].b0_ReadyOn;
Status.ReadyRun := 	SW[1].b1_ReadyRun;
Status.Running := 	SW[1].b2_Running;
Status.Fault := 	SW[1].b3_Fault;
Status.Warning := 	SW[1].b7_Warning;
Status.Remote :=	SW[1].b9_FieldbusCtrlActive;
Status.Commfault :=	Watchdog[1].AlarmAuto;

(*
 * =======================================================================================================================================
 * Translate analog data TO vacon friendly format before sending
 * =======================================================================================================================================
*)

(*Set Values to Vacon*)
FOR i:=1 TO PRG_HMI.DriveSettings.NumberOfDrives BY 1 DO

	(*Set the under/over voltage reference used for load control. Must be between *)
	PDI[i].PDI1_UndervoltageRef := 	REAL_TO_DINT(fun_SafeDivide(divident := PRG_Operation.UnderVoltageRefFiltered_eng, devisor := (PRG_HMI.DriveSettings.NominalDcLinkVoltage/10000)));
	PDI[i].PDI2_OvervoltageRef := 	REAL_TO_DINT(fun_SafeDivide(divident := PRG_Operation.OverVoltageRefFiltered_eng, devisor := (PRG_HMI.DriveSettings.NominalDcLinkVoltage/10000)));

	(*Set the charge or discharge limit between 2% and 100% of the rated source current *)
	PDI[i].PDI3_ChargeLimit := 		LIMIT(20,	REAL_TO_DINT(fun_SafeDivide(divident := PRG_Battery.DriveChargeLimit_eng, devisor := (PRG_HMI.DriveSettings.SourceNomCurrent/1000))), 	1000);
	PDI[i].PDI4_DischargeLimit := 	LIMIT(20,	REAL_TO_DINT(fun_SafeDivide(divident := PRG_Battery.DriveDischargeLimit_eng, devisor := (PRG_HMI.DriveSettings.SourceNomCurrent/1000))), 1000);

	(*Set Min and Max voltage to somewhere between the system's min and max voltage, e.g. 720 and 1008 VDC *)
	PDI[i].PDI5_SourceMaxVoltage := 10*REAL_TO_DINT(PRG_HMI.DriveSettings.SourceMaxVoltage);
	PDI[i].PDI6_SourceMinVoltage := 10*REAL_TO_DINT(PRG_HMI.DriveSettings.SourceMinVoltage);
END_FOR

(*
 * =======================================================================================================================================
 * Prepare digital commands for the control word
 * =======================================================================================================================================
*)

(* Start and stop commands*)
StartStop(
	SET := PRG_StateMain.StartDrive,
	RESET1 := PRG_StateMain.StopDrive OR (PRG_StateMain.tripStatus <> 0)
);

StartTON(
	IN := StartStop.Q1,
	PT := T#500ms
);

(*
 * =======================================================================================================================================
 * Unit over temperature alarm
 * =======================================================================================================================================
*)

UnitOverTempTON(
	IN := Data.UnitTempMax_eng > PRG_HMI.DriveSettings.UnitTempAlarmLevel,
	PT := PRG_HMI.DriveSettings.UnitTempAlarmDelay,
	Q => UnitOverTempAlarm,
	ET =>
);

END_PROGRAM

ACTIONS

END_ACTIONS

(* ---- PRG_Faults.st ---- *)
PROGRAM PRG_Faults
VAR
	BMS_Fault_Word: 			INT := 8; (*Must be first available word number after the ordinary faults*)
	pack: 						INT := 0;
	FaultSR: 					ARRAY[1..20,0..15] OF SR;
	Repeat_Fault: 				fb_RepeatAlarm;
	Reset: 						BOOL;
	CommonAppFault: 			BOOL;
	CommonLevelFault: 			BOOL;
END_VAR

Reset := PRG_Functions.Reset;

CommonAppFault := Repeat_Fault.Alarm_Repeat1 OR Repeat_Fault.Alarm_Repeat3;
CommonLevelFault := Repeat_Fault.Alarm_Repeat2;

(*Common Application Fault*)
FaultSR[1,0] (SET1:=(PRG_BatteryProtection.batteryCommonFault) ,  Q1=>FaultWord[1].0, RESET:=Reset);(*Common Fault from Battery Management System*)
FaultSR[1,1] (SET1:=(NOT PRG_DI.di_FusesOK.PV) ,  Q1=>FaultWord[1].1, RESET:=Reset);(*Line Fuse(s) broken*)
FaultSR[1,2] (SET1:=(NOT PRG_DI.di_LocalEmergencyStop.PV) ,  Q1=>FaultWord[1].2, RESET:=Reset);(*Local Emergency Stop Activated*)
FaultSR[1,3] (SET1:=(NOT PRG_DO.do_ShutdownPlcFailure.PV) ,  Q1=>FaultWord[1].3, RESET:=Reset);(*Fail Safe Shutdown*)
FaultSR[1,4] (SET1:=(NOT PRG_DI.di_DcBreakerEarlyBreak.PV AND PRG_Drive.Status.Running) ,  Q1=>FaultWord[1].4, RESET:=Reset);(*DC Breaker Opened While Running*)
FaultSR[1,5] (SET1:=(PRG_IAS.IAS_FireAlarm) ,  Q1=>FaultWord[1].5, RESET:=Reset);(*Fire Alarm trip from IAS*)
FaultSR[1,6] (SET1:=(PRG_Drive.Status.Fault) ,  Q1=>FaultWord[1].6, RESET:=Reset);(*Vacon Unit -  Common Fault*)
FaultSR[1,7] (SET1:=(PRG_Drive.Status.Commfault) ,  Q1=>FaultWord[1].7, RESET:=Reset);(*Vacon Unit -  Communication Fault*)
FaultSR[1,8] (SET1:=(PRG_Drive.FW2[1].b6_F51_ExternalFault AND PRG_DO.do_ShutdownPlcFailure.PV) ,  Q1=>FaultWord[1].8, RESET:=Reset);(*Remote Emergency Stop*)
FaultSR[1,9] (SET1:=(PRG_BatteryComm.CorvusBMS_Total_Comm_Fault) ,  Q1=>FaultWord[1].9, RESET:=Reset);(*Battery System Total Communication Outage*)
FaultSR[1,10] (SET1:=(NOT PRG_DI.di_RemoteEmergencyStop.PV AND PRG_HMI.enRemoteEstopInput) ,  Q1=>FaultWord[1].10, RESET:=Reset);(*Remote Emergency Stop Activated*)

(*Common Level Fault*)
FaultSR[2,0] (SET1:=(PRG_BatteryProtection.ProtectionTrip_SoC_LL) ,  Q1=>FaultWord[2].0, RESET:=Reset);(*Battery Protection Trip: Low State of Charge*)
FaultSR[2,1] (SET1:=(PRG_BatteryProtection.ProtectionTrip_SoC_HH) ,  Q1=>FaultWord[2].1, RESET:=Reset);(*Battery Protection Trip: High State of Charge*)
FaultSR[2,2] (SET1:=(PRG_BatteryProtection.ProtectionTrip_SoC_LLL) ,  Q1=>FaultWord[2].2, RESET:=Reset);(*Battery Protection Trip: LowLow State of Charge*)
FaultSR[2,3] (SET1:=(PRG_BatteryProtection.ProtectionTrip_Undervoltage) ,  Q1=>FaultWord[2].3, RESET:=Reset);(*Battery Protection Trip: Low Battery Voltage*)
FaultSR[2,4] (SET1:=(PRG_BatteryProtection.ProtectionTrip_Overvoltage) ,  Q1=>FaultWord[2].4, RESET:=Reset);(*Battery Protection Trip: High Battery Voltage*)
FaultSR[2,5] (SET1:=(PRG_BatteryProtection.ProtectionTrip_CellVolt_HH) ,  Q1=>FaultWord[2].5, RESET:=Reset);(*Battery Protection Trip: High Cell Voltage*)
FaultSR[2,6] (SET1:=(PRG_BatteryProtection.ProtectionTrip_CellVolt_LL) ,  Q1=>FaultWord[2].6, RESET:=Reset);(*Battery Protection Trip: Low Cell Voltage*)
FaultSR[2,7] (SET1:=(PRG_BatteryProtection.ProtectionTrip_CellTemp_HH) ,  Q1=>FaultWord[2].7, RESET:=Reset);(*Battery Protection Trip: High Cell Temperature*)
FaultSR[2,8] (SET1:=(PRG_AI.ai_FilterTemperature.Alarm.HHH) ,  Q1=>FaultWord[2].8, RESET:=Reset);(*Filter Temperature High High*)

(*Vacon Drive Faults*)
FaultSR[3,0] (SET1:=(PRG_Drive.FW[1].b0_F1_Overcurrent) ,  Q1=>FaultWord[3].0, RESET:=Reset);(*Vacon Unit -  Over Current Fault*)
FaultSR[3,1] (SET1:=(PRG_Drive.FW[1].b1_F2_OverVoltage) ,  Q1=>FaultWord[3].1, RESET:=Reset);(*Vacon Unit -  Over Voltage Fault*)
FaultSR[3,2] (SET1:=(PRG_Drive.FW[1].b2_F9_UnderVoltage) ,  Q1=>FaultWord[3].2, RESET:=Reset);(*Vacon Unit -  Under Voltage Fault*)
FaultSR[3,3] (SET1:=(PRG_Drive.FW[1].b4_F3_EarthFaultDrive) ,  Q1=>FaultWord[3].3, RESET:=Reset);(*Vacon Unit -  Earth Fault*)
FaultSR[3,4] (SET1:=(PRG_Drive.FW[1].b6_F14_UnitOverTemp) ,  Q1=>FaultWord[3].4, RESET:=Reset);(*Vacon Unit -  Over Temperature Fault*)
FaultSR[3,5] (SET1:=(PRG_Drive.FW[1].b7_F29_ThermistorFault) ,  Q1=>FaultWord[3].5, RESET:=Reset);(*Vacon Unit -  Temperature Measurement Fault*)
FaultSR[3,6] (SET1:=(PRG_Drive.FW[1].b11_F52_KeypadCommFault) ,  Q1=>FaultWord[3].6, RESET:=Reset);(*Vacon Unit -  Keypad Communication Fault*)
FaultSR[3,7] (SET1:=(PRG_Drive.FW[1].b12_F53_FieldbusCommFault) ,  Q1=>FaultWord[3].7, RESET:=Reset);(*Vacon Unit -  Fieldbus Communication Fault*)
FaultSR[3,8] (SET1:=(PRG_Drive.FW[1].b14_F54_SlotCommFault) ,  Q1=>FaultWord[3].8, RESET:=Reset);(*Vacon Unit -  Expansion Slot Communication Fault*)
FaultSR[3,9] (SET1:=(PRG_Drive.FW[1].b15_F50_4mAFault) ,  Q1=>FaultWord[3].9, RESET:=Reset);(*Vacon Unit -  4 mA Fault*)

(*Auto generated alarms from Corvus BMS*)
BMS_Fault_Word := 4; (*Next available faultword*)
FOR pack := 1 TO PRG_HMI.setup_Battery_total_nr_of_packs BY 1 DO
	FaultSR[BMS_Fault_Word,0] (SET1 := (PRG_BatteryComm.CorvusRead[pack].FW.Contactor_Fault), Q1 => FaultWord[BMS_Fault_Word].0, RESET := Reset); 					(*BMS Pack Contactor Fault*)
	FaultSR[BMS_Fault_Word,1] (SET1 := (PRG_BatteryComm.CorvusRead[pack].FW.Deep_OverDischarge_Lockout_Fault), Q1 => FaultWord[BMS_Fault_Word].1, RESET := Reset); 	(*BMS Pack Over Discharge Lockout Fault*)
	FaultSR[BMS_Fault_Word,2] (SET1 := (PRG_BatteryComm.CorvusRead[pack].FW.E_Stop_Active_Fault), Q1 => FaultWord[BMS_Fault_Word].2, RESET := Reset); 				(*BMS Pack E-stop Active*)
	FaultSR[BMS_Fault_Word,3] (SET1 := (PRG_BatteryComm.CorvusRead[pack].FW.Ground_Fault), Q1 => FaultWord[BMS_Fault_Word].3, RESET := Reset); 						(*BMS Pack Ground Fault*)
	FaultSR[BMS_Fault_Word,4] (SET1 := (PRG_BatteryComm.CorvusRead[pack].FW.HVIL_Fault), Q1 => FaultWord[BMS_Fault_Word].4, RESET := Reset); 							(*BMS Pack High Voltage Interlock Loop Open*)
	FaultSR[BMS_Fault_Word,5] (SET1 := (PRG_BatteryComm.CorvusRead[pack].FW.Low_Temp_OverCurrent_Fault), Q1 => FaultWord[BMS_Fault_Word].5, RESET := Reset); 			(*BMS Pack Low Temp. Over Current Fault*)
	FaultSR[BMS_Fault_Word,6] (SET1 := (PRG_BatteryComm.CorvusRead[pack].FW.PDM_OverTemperature_Fault), Q1 => FaultWord[BMS_Fault_Word].6, RESET := Reset); 			(*BMS Pack Over Temperature Fault*)
	FaultSR[BMS_Fault_Word,7] (SET1 := (PRG_BatteryComm.CorvusRead[pack].FW.Repeated_OverCharge_Lockout_Fault), Q1 => FaultWord[BMS_Fault_Word].7, RESET := Reset); 	(*BMS Pack Over Charge Lockout Fault*)
	FaultSR[BMS_Fault_Word,8] (SET1 := (PRG_BatteryComm.CorvusRead[pack].FW.Safety_Shutdown_Fault), Q1 => FaultWord[BMS_Fault_Word].8, RESET := Reset); 				(*BMS Pack Safety Shutdown Fault*)
	FaultSR[BMS_Fault_Word,9] (SET1 := (PRG_BatteryComm.CorvusRead[pack].FW.SE_overTemperature_Fault), Q1 => FaultWord[BMS_Fault_Word].9, RESET := Reset); 			(*BMS Pack Cell Over Temperature Fault*)
	FaultSR[BMS_Fault_Word,10] (SET1 := (PRG_BatteryComm.CorvusRead[pack].FW.SE_overVoltage_Fault), Q1 => FaultWord[BMS_Fault_Word].10, RESET := Reset); 				(*BMS Pack Cell Over Voltage Fault*)
	FaultSR[BMS_Fault_Word,11] (SET1 := (PRG_BatteryComm.CorvusRead[pack].FW.SE_underVoltage_Fault), Q1 => FaultWord[BMS_Fault_Word].11, RESET:=Reset);				(*BMS Pack Cell Under Voltage Fault*)
	BMS_Fault_Word :=  BMS_Fault_Word+1;
END_FOR

(*Blinks the alarm output*)

Repeat_Fault(
	AlarmWord1:= INT_TO_WORD(FaultWord[1]),
	AlarmWord2:= INT_TO_WORD(FaultWord[2]),
	AlarmWord3:= INT_TO_WORD(FaultWord[3]),
	AlarmWord4:= INT_TO_WORD(FaultWord[4]),
	AlarmWord5:= INT_TO_WORD(FaultWord[5]),
	AlarmWord6:= INT_TO_WORD(FaultWord[6]),
	AlarmWord7:= INT_TO_WORD(FaultWord[7]),
	AlarmWord8:= INT_TO_WORD(FaultWord[8]),
	AlarmWord9:= INT_TO_WORD(FaultWord[9]),
	AlarmWord10:= INT_TO_WORD(FaultWord[10]),
	AlarmWord11:= INT_TO_WORD(FaultWord[11]),
	AlarmWord12:= INT_TO_WORD(FaultWord[12]),
	AlarmWord13:= INT_TO_WORD(FaultWord[13]),
	AlarmWord14:= INT_TO_WORD(FaultWord[14]),
	AlarmWord15:= INT_TO_WORD(FaultWord[15]),
	AlarmWord16:= INT_TO_WORD(FaultWord[16]),
	AlarmWord17:= INT_TO_WORD(FaultWord[17]),
	AlarmWord18:= INT_TO_WORD(FaultWord[18]),
	AlarmWord19:= INT_TO_WORD(FaultWord[19]),
	AlarmWord20:= INT_TO_WORD(FaultWord[20]),
	Alarm_common => ,
	Alarm_count => ,
	Alarm_Repeat1 => ,
	Alarm_Repeat2 => ,
	Alarm_Repeat3 => ,
	Alarm_Repeat4 => ,
	Alarm_Repeat5 => ,
	Alarm_Repeat6 => ,
	Alarm_Repeat7 => ,
	Alarm_Repeat8 => ,
	Alarm_Repeat9 => ,
	Alarm_Repeat10 => ,
	Alarm_Repeat11 => ,
	Alarm_Repeat12 => ,
	Alarm_Repeat13 => ,
	Alarm_Repeat14 => ,
	Alarm_Repeat15 => ,
	Alarm_Repeat16 => ,
	Alarm_Repeat17 => ,
	Alarm_Repeat18 => ,
	Alarm_Repeat19 => ,
	Alarm_Repeat20 =>
);

END_PROGRAM

ACTIONS
ACTION hmi_Faults
hmi_FaultWord[1].0 := FaultSR[1,0].Q1;
hmi_FaultWord[1].1 := FaultSR[1,1].Q1;
hmi_FaultWord[1].2 := FaultSR[1,2].Q1;
hmi_FaultWord[1].3 := FaultSR[1,3].Q1;
hmi_FaultWord[1].4 := FaultSR[1,4].Q1;
hmi_FaultWord[1].5 := FaultSR[1,5].Q1;
hmi_FaultWord[1].6 := FaultSR[1,6].Q1;
hmi_FaultWord[1].7 := FaultSR[1,7].Q1;
hmi_FaultWord[1].8 := FaultSR[1,8].Q1;
hmi_FaultWord[1].9 := FaultSR[1,9].Q1;
hmi_FaultWord[1].10 := FaultSR[1,10].Q1;
hmi_FaultWord[1].11 := FaultSR[1,11].Q1;
hmi_FaultWord[1].12 := FaultSR[1,12].Q1;
hmi_FaultWord[1].13 := FaultSR[1,13].Q1;
hmi_FaultWord[1].14 := FaultSR[1,14].Q1;
hmi_FaultWord[1].15 := FaultSR[1,15].Q1;
hmi_FaultWord[2].0 := FaultSR[2,0].Q1;
hmi_FaultWord[2].1 := FaultSR[2,1].Q1;
hmi_FaultWord[2].2 := FaultSR[2,2].Q1;
hmi_FaultWord[2].3 := FaultSR[2,3].Q1;
hmi_FaultWord[2].4 := FaultSR[2,4].Q1;
hmi_FaultWord[2].5 := FaultSR[2,5].Q1;
hmi_FaultWord[2].6 := FaultSR[2,6].Q1;
hmi_FaultWord[2].7 := FaultSR[2,7].Q1;
hmi_FaultWord[2].8 := FaultSR[2,8].Q1;
hmi_FaultWord[2].9 := FaultSR[2,9].Q1;
hmi_FaultWord[2].10 := FaultSR[2,10].Q1;
hmi_FaultWord[2].11 := FaultSR[2,11].Q1;
hmi_FaultWord[2].12 := FaultSR[2,12].Q1;
hmi_FaultWord[2].13 := FaultSR[2,13].Q1;
hmi_FaultWord[2].14 := FaultSR[2,14].Q1;
hmi_FaultWord[2].15 := FaultSR[2,15].Q1;
hmi_FaultWord[3].0 := FaultSR[3,0].Q1;
hmi_FaultWord[3].1 := FaultSR[3,1].Q1;
hmi_FaultWord[3].2 := FaultSR[3,2].Q1;
hmi_FaultWord[3].3 := FaultSR[3,3].Q1;
hmi_FaultWord[3].4 := FaultSR[3,4].Q1;
hmi_FaultWord[3].5 := FaultSR[3,5].Q1;
hmi_FaultWord[3].6 := FaultSR[3,6].Q1;
hmi_FaultWord[3].7 := FaultSR[3,7].Q1;
hmi_FaultWord[3].8 := FaultSR[3,8].Q1;
hmi_FaultWord[3].9 := FaultSR[3,9].Q1;
hmi_FaultWord[3].10 := FaultSR[3,10].Q1;
hmi_FaultWord[3].11 := FaultSR[3,11].Q1;
hmi_FaultWord[3].12 := FaultSR[3,12].Q1;
hmi_FaultWord[3].13 := FaultSR[3,13].Q1;
hmi_FaultWord[3].14 := FaultSR[3,14].Q1;
hmi_FaultWord[3].15 := FaultSR[3,15].Q1;
hmi_FaultWord[4].0 := FaultSR[4,0].Q1;
hmi_FaultWord[4].1 := FaultSR[4,1].Q1;
hmi_FaultWord[4].2 := FaultSR[4,2].Q1;
hmi_FaultWord[4].3 := FaultSR[4,3].Q1;
hmi_FaultWord[4].4 := FaultSR[4,4].Q1;
hmi_FaultWord[4].5 := FaultSR[4,5].Q1;
hmi_FaultWord[4].6 := FaultSR[4,6].Q1;
hmi_FaultWord[4].7 := FaultSR[4,7].Q1;
hmi_FaultWord[4].8 := FaultSR[4,8].Q1;
hmi_FaultWord[4].9 := FaultSR[4,9].Q1;
hmi_FaultWord[4].10 := FaultSR[4,10].Q1;
hmi_FaultWord[4].11 := FaultSR[4,11].Q1;
hmi_FaultWord[4].12 := FaultSR[4,12].Q1;
hmi_FaultWord[4].13 := FaultSR[4,13].Q1;
hmi_FaultWord[4].14 := FaultSR[4,14].Q1;
hmi_FaultWord[4].15 := FaultSR[4,15].Q1;
hmi_FaultWord[5].0 := FaultSR[5,0].Q1;
hmi_FaultWord[5].1 := FaultSR[5,1].Q1;
hmi_FaultWord[5].2 := FaultSR[5,2].Q1;
hmi_FaultWord[5].3 := FaultSR[5,3].Q1;
hmi_FaultWord[5].4 := FaultSR[5,4].Q1;
hmi_FaultWord[5].5 := FaultSR[5,5].Q1;
hmi_FaultWord[5].6 := FaultSR[5,6].Q1;
hmi_FaultWord[5].7 := FaultSR[5,7].Q1;
hmi_FaultWord[5].8 := FaultSR[5,8].Q1;
hmi_FaultWord[5].9 := FaultSR[5,9].Q1;
hmi_FaultWord[5].10 := FaultSR[5,10].Q1;
hmi_FaultWord[5].11 := FaultSR[5,11].Q1;
hmi_FaultWord[5].12 := FaultSR[5,12].Q1;
hmi_FaultWord[5].13 := FaultSR[5,13].Q1;
hmi_FaultWord[5].14 := FaultSR[5,14].Q1;
hmi_FaultWord[5].15 := FaultSR[5,15].Q1;
hmi_FaultWord[6].0 := FaultSR[6,0].Q1;
hmi_FaultWord[6].1 := FaultSR[6,1].Q1;
hmi_FaultWord[6].2 := FaultSR[6,2].Q1;
hmi_FaultWord[6].3 := FaultSR[6,3].Q1;
hmi_FaultWord[6].4 := FaultSR[6,4].Q1;
hmi_FaultWord[6].5 := FaultSR[6,5].Q1;
hmi_FaultWord[6].6 := FaultSR[6,6].Q1;
hmi_FaultWord[6].7 := FaultSR[6,7].Q1;
hmi_FaultWord[6].8 := FaultSR[6,8].Q1;
hmi_FaultWord[6].9 := FaultSR[6,9].Q1;
hmi_FaultWord[6].10 := FaultSR[6,10].Q1;
hmi_FaultWord[6].11 := FaultSR[6,11].Q1;
hmi_FaultWord[6].12 := FaultSR[6,12].Q1;
hmi_FaultWord[6].13 := FaultSR[6,13].Q1;
hmi_FaultWord[6].14 := FaultSR[6,14].Q1;
hmi_FaultWord[6].15 := FaultSR[6,15].Q1;
hmi_FaultWord[7].0 := FaultSR[7,0].Q1;
hmi_FaultWord[7].1 := FaultSR[7,1].Q1;
hmi_FaultWord[7].2 := FaultSR[7,2].Q1;
hmi_FaultWord[7].3 := FaultSR[7,3].Q1;
hmi_FaultWord[7].4 := FaultSR[7,4].Q1;
hmi_FaultWord[7].5 := FaultSR[7,5].Q1;
hmi_FaultWord[7].6 := FaultSR[7,6].Q1;
hmi_FaultWord[7].7 := FaultSR[7,7].Q1;
hmi_FaultWord[7].8 := FaultSR[7,8].Q1;
hmi_FaultWord[7].9 := FaultSR[7,9].Q1;
hmi_FaultWord[7].10 := FaultSR[7,10].Q1;
hmi_FaultWord[7].11 := FaultSR[7,11].Q1;
hmi_FaultWord[7].12 := FaultSR[7,12].Q1;
hmi_FaultWord[7].13 := FaultSR[7,13].Q1;
hmi_FaultWord[7].14 := FaultSR[7,14].Q1;
hmi_FaultWord[7].15 := FaultSR[7,15].Q1;
hmi_FaultWord[8].0 := FaultSR[8,0].Q1;
hmi_FaultWord[8].1 := FaultSR[8,1].Q1;
hmi_FaultWord[8].2 := FaultSR[8,2].Q1;
hmi_FaultWord[8].3 := FaultSR[8,3].Q1;
hmi_FaultWord[8].4 := FaultSR[8,4].Q1;
hmi_FaultWord[8].5 := FaultSR[8,5].Q1;
hmi_FaultWord[8].6 := FaultSR[8,6].Q1;
hmi_FaultWord[8].7 := FaultSR[8,7].Q1;
hmi_FaultWord[8].8 := FaultSR[8,8].Q1;
hmi_FaultWord[8].9 := FaultSR[8,9].Q1;
hmi_FaultWord[8].10 := FaultSR[8,10].Q1;
hmi_FaultWord[8].11 := FaultSR[8,11].Q1;
hmi_FaultWord[8].12 := FaultSR[8,12].Q1;
hmi_FaultWord[8].13 := FaultSR[8,13].Q1;
hmi_FaultWord[8].14 := FaultSR[8,14].Q1;
hmi_FaultWord[8].15 := FaultSR[8,15].Q1;
hmi_FaultWord[9].0 := FaultSR[9,0].Q1;
hmi_FaultWord[9].1 := FaultSR[9,1].Q1;
hmi_FaultWord[9].2 := FaultSR[9,2].Q1;
hmi_FaultWord[9].3 := FaultSR[9,3].Q1;
hmi_FaultWord[9].4 := FaultSR[9,4].Q1;
hmi_FaultWord[9].5 := FaultSR[9,5].Q1;
hmi_FaultWord[9].6 := FaultSR[9,6].Q1;
hmi_FaultWord[9].7 := FaultSR[9,7].Q1;
hmi_FaultWord[9].8 := FaultSR[9,8].Q1;
hmi_FaultWord[9].9 := FaultSR[9,9].Q1;
hmi_FaultWord[9].10 := FaultSR[9,10].Q1;
hmi_FaultWord[9].11 := FaultSR[9,11].Q1;
hmi_FaultWord[9].12 := FaultSR[9,12].Q1;
hmi_FaultWord[9].13 := FaultSR[9,13].Q1;
hmi_FaultWord[9].14 := FaultSR[9,14].Q1;
hmi_FaultWord[9].15 := FaultSR[9,15].Q1;
hmi_FaultWord[10].0 := FaultSR[10,0].Q1;
hmi_FaultWord[10].1 := FaultSR[10,1].Q1;
hmi_FaultWord[10].2 := FaultSR[10,2].Q1;
hmi_FaultWord[10].3 := FaultSR[10,3].Q1;
hmi_FaultWord[10].4 := FaultSR[10,4].Q1;
hmi_FaultWord[10].5 := FaultSR[10,5].Q1;
hmi_FaultWord[10].6 := FaultSR[10,6].Q1;
hmi_FaultWord[10].7 := FaultSR[10,7].Q1;
hmi_FaultWord[10].8 := FaultSR[10,8].Q1;
hmi_FaultWord[10].9 := FaultSR[10,9].Q1;
hmi_FaultWord[10].10 := FaultSR[10,10].Q1;
hmi_FaultWord[10].11 := FaultSR[10,11].Q1;
hmi_FaultWord[10].12 := FaultSR[10,12].Q1;
hmi_FaultWord[10].13 := FaultSR[10,13].Q1;
hmi_FaultWord[10].14 := FaultSR[10,14].Q1;
hmi_FaultWord[10].15 := FaultSR[10,15].Q1;

END_ACTION
END_ACTIONS

(* ---- PRG_Functions.st ---- *)
PROGRAM PRG_Functions
VAR
	(*Reset Function*)
	ResetTOF :	TOF;
	Reset: BOOL;

	(*Breaker position*)
	Breaker : fb_DiDiVerif;
	Version: 				fb_VersionRead;
	ProjectVersion: 		STRING(60);

	(*Time synch*)
	TimeSynch : fb_remoteTime;

	(*Export Retain Data*)
	RetainExport : 			Smi_RetainExport;	(*Function block for saving retain data to XML*)
	RetainExportRT :		R_TRIG;				(*Trigger export of retain data*)
	DateTime :				TIMESPEC;			(*The PLCs real time clock and date*)
	Filename :				STRING(100);		(*File name, including full path, for retain export*)
	Filedate :				STRING(30);			(*File date for automatic file name when saving retain memory*)
	RetainState:			DINT;				(*State of retain saving process*)
	RetainError:			BOOL;				(*If retain can not be saved*)
	ModuleData :			TCS_ARGINFO;		(*Get some information about the plc*)
	InstanceName :			STRING(15);			(*Instance name in software module list - used for filename*)

	FirstRun: 				BOOL := 0;
	LastCommit: 			fb_LastCommit;
END_VAR

(*
 * =======================================================================================================================================
 * Reset Function
 * =======================================================================================================================================
*)
ResetTOF(
	IN := (PRG_DI.di_LocalReset.PV
	 OR PRG_IAS.IAS_CTRL_Commands.5
	 OR PRG_HMI.Reset
	 OR PRG_StateMain.State = e_Init
	),
	PT := T#5000ms
);

Reset := ResetTOF.Q AND PRG_StateMain.LedBlink;

(*
 * =======================================================================================================================================
 * Breaker Position
 * =======================================================================================================================================
*)

Breaker(
	Reset := Reset,
	DI_1_NC := PRG_DI.di_DcBreakerClosed.PV,
	DI_2_NO := PRG_DI.di_DcBreakerOpen.PV,
	Inhibit_alarm := FALSE,
	Alarm_delay := T#1s,
	Verif_delay := T#0.5s,
	Alarm_inst => ,
	Alarm_delayed => ,
	DI_Verif_delay => ,
	DI_Verif =>
);

(*
 * =======================================================================================================================================
 * Project Version
 * =======================================================================================================================================
*)
Version(
	VersionRead :=  PRG_StateMain.State = e_Init OR Reset,
	CommitHash := LastCommit.LastCommitShort
);

(*
 * =======================================================================================================================================
 * Read git repository commit hash
 * =======================================================================================================================================
*)
LastCommit;

(*
 * =======================================================================================================================================
 * Time Synch from IAS
 * =======================================================================================================================================
*)

TimeSynch(
	EN := NOT PRG_IAS.IasCommunication.Alarm,
	Hour := PRG_IAS.IAS_CTRL_Hours,
	Minute := PRG_IAS.IAS_CTRL_Minutes,
	Second := PRG_IAS.IAS_CTRL_Seconds,
	dtTime => ,
	plcTime =>
);

(*
 * =======================================================================================================================================
 * Export retain memory into file
 * =======================================================================================================================================
*)

(*Manual export command from HMI*)
RetainExportRT(CLK := PRG_HMI.RetainExportCmd, Q => );

(*Find date and create file name*)
IF RetainExportRT.Q OR NOT FirstRun THEN
	ModuleData := Tcs_ARG_GetConfig(Dummy := 0);
	InstanceName := ModuleData.Name;	(*Same as module instance name in Software-section in Solution center tree*)
	DateTime :=  RTC_GetClock(dummy := FALSE);
	Filedate := LEFT(RIGHT(STR:=DT_TO_STRING(DateTime.DateAndTime),SIZE:=19 ),10);	(*Format: 2018-12-24*)

	(*Build full path and file name for saving the XML file*)
	Filename := '/cfc0/RetainExport/';				(*Save folder*)
	Filename := CONCAT(Filename, InstanceName);		(*Add file name, it starts with the software module instance name*)
	IF RetainExportRT.Q THEN 						(*If manual creation - Add today's date*)
		Filename := CONCAT(Filename, '-');			(*Add a dash before date*)
		Filename := CONCAT(Filename, Filedate);		(*Add date*)
	ELSE 											(*If autosaved on first run, then postfix that the file is autosaved.*)
		Filename := CONCAT(Filename, '-Autosaved');	(* No date as we want the file to be overwritten at each firstrun*)
	END_IF
	Filename := CONCAT(Filename, '.xml');			(*add file format*)
END_IF

(*Do the actual export*)
RetainExport(
	Request := RetainExportRT.Q OR NOT FirstRun,
	FileName := Filename,
	State => RetainState,
	Error => RetainError
);

(*Set flag so that firstrun is not same as secondrun :) *)
FirstRun := TRUE;

END_PROGRAM
